PROGRAM MAIN
VAR
END_VAR

END_PROGRAM

(* stored: Version 1.1.0.1
   POU MAIN: Id {377dca09-b62a-4413-b1d6-b874157f8cb8} *)
